// TIA Portal V17 export
// export: Created 2025-06-26T07:49:55.3606445Z, ExportSetting WithDefaults, DisplayName Totally Integrated Automation Portal, DisplayVersion V17 Update 8, DisplayName TIA Portal Openness, DisplayVersion V17 Update 8, DisplayName TIA Portal Version Control Interface, DisplayVersion V17, DisplayName STEP 7 Professional, DisplayVersion V17 Update 8, DisplayName STEP 7 Safety, DisplayVersion V17 Update 6, DisplayName WinCC Advanced, DisplayVersion V17 Update 8
TYPE "stCirculationPump"
// stored: IsFailsafeCompliant false
   STRUCT
      bEnable : Bool;   // 1 = enabled 0 = disabled
      bManualMode : Bool;   // 1 = manual, 0 = auto
      bManualRun : Bool;   // 1 = force run, 0 = off
      bOutput : Bool;   // 1 = run, 0 = stop
      bFault : Bool;   // 1 = fault, 0 = ok
      bPressureLow : Bool;   // 1 = pressure low, 0 = ok
      bTemperatureHigh : Bool;   // 1 = temperature high, 0 = ok
      bDifferentialPressureHigh : Bool;   // 1 = pressure high, 0 = ok
      bReservoirLow : Bool;   // 1 = reservoir low, 0 = ok
      bDeltaTHigh : Bool;   // 1 = delta T high, 0 = ok
      bPressureHigh : Bool;   // 1 = pressure high, 0 = ok
      nMode : USInt;   // 0 = Off, 1 = Auto, 2 = Manual
   END_STRUCT;
END_TYPE
